{attribute 'linkalways'} 
{attribute 'no_explicit_call' := 'This FB is a CLASS and must be accessed using methods or properties'}
{attribute 'enable_dynamic_creation'}
FUNCTION_BLOCK _ETcVnLineType EXTENDS EnumDatatypeBase
VAR
	localData : ETcVnLineType;
	activeData : REFERENCE TO ETcVnLineType;
	enumBaseDatatype : _DINT(localData);
END_VAR

METHOD PRIVATE AddLocalEnumeration
VAR_INPUT
	Enumeration : T_MAXSTRING;
	Value : ETcVnLineType;
END_VAR
AddEnumeration(Enumeration, Value);
END_METHOD

PROPERTY PUBLIC Address : PVOID
GET
Address := ADR(activeData);
END_GET
END_PROPERTY

METHOD PUBLIC ClearReference
VAR_INPUT
END_VAR
activeData REF= localData;
SetBaseDatatypeReference();
END_METHOD

METHOD PUBLIC Clone : I_Datatype
VAR
    pClone : POINTER TO _ETcVnLineType;
END_VAR
pClone := __NEW(_ETcVnLineType(InitialValue := Value));
Clone := pClone^;
END_METHOD

METHOD FB_init : BOOL
VAR_INPUT
	bInitRetains : BOOL; // if TRUE, the retain variables are initialized (warm start / cold start)
	bInCopyCode : BOOL;  // if TRUE, the instance afterwards gets moved into the copy code (online change)
	InitialValue : ETcVnLineType;
END_VAR
localData := InitialValue;
AddBaseDatatype(enumBaseDatatype);
ClearReference();

AddLocalEnumeration('TCVN_LT_4_CONNECTED', ETcVnLineType.TCVN_LT_4_CONNECTED);
AddLocalEnumeration('TCVN_LT_8_CONNECTED', ETcVnLineType.TCVN_LT_8_CONNECTED);
AddLocalEnumeration('TCVN_LT_ANTIALIASED', ETcVnLineType.TCVN_LT_ANTIALIASED);
END_METHOD

PROPERTY PUBLIC Identifier : T_MAXSTRING
GET
Identifier := 'ETcVnLineType';
END_GET
END_PROPERTY

METHOD IsEnumeratorValueEqual : BOOL
VAR_INPUT
	Enumerator : I_KeyValueForwardEnumerator;
END_VAR
VAR
	storedValue : ETcVnLineType;
END_VAR
IF NOT Enumerator.TryGet(storedValue) THEN
	RETURN;
END_IF

IsEnumeratorValueEqual := storedValue = activeData;
END_METHOD

METHOD PUBLIC MakeReferenceTo
VAR_INPUT
	ReferenceTarget : REFERENCE TO ETcVnLineType;
END_VAR
activeData REF= ReferenceTarget;
SetBaseDatatypeReference();
END_METHOD

METHOD PROTECTED SetBaseDatatypeReference
VAR_INPUT
END_VAR
enumBaseDatatype.MakeReferenceTo(activeData);
END_METHOD

PROPERTY PUBLIC Size : UDINT
GET
Size := SIZEOF(activeData);
END_GET
END_PROPERTY

METHOD TryMakeReferenceTo : BOOL
VAR_INPUT
	Target : I_Datatype;
END_VAR
VAR
	targetAsEnum : I_EnumDatatype;
	pTargetData : POINTER TO ETcVnLineType;
END_VAR
IF NOT Target.TryResolveAsEnumDatatype(targetAsEnum) THEN
	RETURN;
END_IF

IF targetAsEnum.Identifier <> Identifier THEN
	RETURN;
END_IF

pTargetData := Target.Address;
activeData REF= pTargetData^;
SetBaseDatatypeReference();
TryMakeReferenceTo := TRUE;
END_METHOD

PROPERTY PUBLIC Value : ETcVnLineType
GET
Value := activeData;
END_GET
SET
activeData := Value;
END_SET
END_PROPERTY

END_FUNCTION_BLOCK

(* stored: Version 1.1.0.1, ProductVersion 3.1.4024.12
   POU _ETcVnLineType: Id {a32b0db0-3577-4253-9f77-9c5496d99624}, SpecialFunc None
   Folder Constructor: Id {69f70c9b-a0cd-4028-852c-aecba2493ab7}
   Folder Private: Id {f978207c-8f4f-45a6-a57f-43f3f96e4d00}
   Folder Protected: Id {cca43355-0a5a-4f91-a4cc-c93384204700}
   Method AddLocalEnumeration: Id {685cd485-2183-4a54-a8b6-53b181f8799f}
   Property Address: Id {738d668a-d34e-4c6c-8142-318c992a545b}
   Get Get: Id {40df5a0f-6823-47f2-9f55-4e290e4e3b9b}
   Method ClearReference: Id {e91b8e52-2d6c-4b2c-abaf-88e17152b4b5}
   Method Clone: Id {c26ffb68-3a90-4bfd-a3e2-b4fb71fad3ab}
   Method FB_init: Id {bcc53c76-c207-42c1-b33e-f0e35c684881}
   Property Identifier: Id {1fdb4395-606e-4042-8bbb-e1aed41f87ac}
   Get Get: Id {2c4fe9a2-5c4e-432b-8640-7d0a4e1d07f7}
   Method IsEnumeratorValueEqual: Id {b542f196-3858-47f7-84c0-bb71eebcd051}
   Method MakeReferenceTo: Id {6de11e62-45c2-467e-be18-671ecd1cc82c}
   Method SetBaseDatatypeReference: Id {c5615976-4750-479b-8d52-0ce4b027ca8d}
   Property Size: Id {a886569f-b8f7-4dd6-8078-20713c74c00d}
   Get Get: Id {ad34fe1a-8bdc-4ef6-afc9-beca72941ffe}
   Method TryMakeReferenceTo: Id {568fcff7-ed75-42b3-ac41-a7c72b248feb}
   Property Value: Id {30a718f5-e319-49a6-9e9b-1531448f60bf}
   Get Get: Id {519ec237-f63c-4c35-8903-35553216c156}
   Set Set: Id {40a310f0-cd2f-4381-8ea7-81b2f16c3d0b} *)
